# EPICS substitutions: LukasWaveformReaderApp/Db/waveform.substitutions
#Substitution file

file waveform.template
{
pattern
{channel}
{"0"}
{"1"}
{"2"}
{"3"}
{"4"}
{"5"}
}
